INTERFACE I_QueueNode

PROPERTY PUBLIC DataType : T_MaxString
GET
END_GET
END_PROPERTY

METHOD PUBLIC Destroy
VAR_INPUT
END_VAR
END_METHOD

METHOD PUBLIC Get : BOOL;
VAR_INPUT
	Destination : ANY;
END_VAR
END_METHOD

PROPERTY PUBLIC Next : I_QueueNode
GET
END_GET
SET
END_SET
END_PROPERTY

END_INTERFACE

(* stored: Version 1.1.0.1, ProductVersion 3.1.4024.11
   Itf I_QueueNode: Id {6b75ffa8-a79b-4321-92d0-ec8c46d024a4}
   Property DataType: Id {6b8d9287-5a35-48a2-b3ff-1f347497c788}
   Get Get: Id {530f547b-5527-442c-9dc2-d053441fdf66}
   Method Destroy: Id {f562c5a5-3c44-4553-882f-168d43d6e471}
   Method Get: Id {2ff680fb-9677-474d-b509-5468772db183}
   Property Next: Id {00d54bf8-d054-45d2-894d-565e6e8eb72c}
   Get Get: Id {aa775674-5714-49ad-855b-fbddd8492b66}
   Set Set: Id {37c75405-a241-4f41-8f32-04a8c89d1da6} *)
